FUNCTION_BLOCK FB_Syntax_ExhaustiveArraysAndFBInit
VAR
    // --- 1. Basic & Multi-dimensional Arrays ---
    arr1DPrimitives      : ARRAY[1..5] OF INT := [10, 20, 30, 40, 50];
    arr1DMultilineMatrix : ARRAY[1..12] OF INT := [
        1, 2, 3, 4,
        5, 6, 7, 8,
        9, 10, 11, 12
    ];
    arr2DMatrix : ARRAY[1..3, 1..4] OF INT;
    arr3DCube   : ARRAY[0..1, 0..1, 0..1] OF BOOL;
    arr4DHyper  : ARRAY[1..2, 1..2, 1..2, 1..2] OF BYTE;

    // --- 2. Negative, Zero-based, and Subrange Bounds ---
    arrNegativeBounds : ARRAY[-5..5] OF INT     := [-5, -4, -3, -2, -1, 0, 1, 2, 3, 4, 5];
    arrOffsetBounds   : ARRAY[100..105] OF DINT := [1000, 1001, 1002, 1003, 1004, 1005];

    // --- 3. Repetition / Initialization Factors ---
    arrRepeatZeros  : ARRAY[1..100] OF INT      := [100(0)];
    arrRepeatMixed  : ARRAY[1..10] OF INT       := [5(15), 3(25), 2(0)];
    arrRepeatString : ARRAY[1..4] OF STRING(30) := [2('READY'), 2('ERROR')];

    // --- 4. Arrays of STRUCT / UDT ---
    arrStructSingleLine     : ARRAY[1..4] OF ST_Syntax_Mini := [
        (nId := 1, bActive := TRUE, sName := 'Stage-Inlet'),
        (nId := 2, bActive := TRUE, sName := 'Stage-Reaction'),
        (nId := 3, bActive := TRUE, sName := 'Stage-Separation'),
        (nId := 4, bActive := TRUE, sName := 'Stage-Outlet')
    ];
    arrStructExpanded       : ARRAY[1..2] OF ST_Syntax_Mini := [
        (
            nId     := 101,
            bActive := TRUE,
            sName   := 'NodeA'
        ),
        (
            nId     := 102,
            bActive := FALSE,
            sName   := 'NodeB'
        )
    ];

    // --- 5. Arrays of Function Blocks with FB_init Parameters ---
    arrFbInitSingleLine : ARRAY[1..2] OF FB_Syntax_FBInitMethods[(nInitialId := 1, sInitialName := 'MotorA'), (nInitialId := 2, sInitialName := 'MotorB')];
    arrFbInitMultiline  : ARRAY[1..2] OF FB_Syntax_FBInitMethods[(nInitialId := 10, sInitialName := 'Sensor_Primary'), (nInitialId := 20, sInitialName := 'Sensor_Secondary')];

    // --- 6. Arrays of POINTER TO and INTERFACE ---
    arrPointers       : ARRAY[1..4] OF POINTER TO DINT;
    arrStructPointers : ARRAY[1..4] OF POINTER TO ST_Syntax_Mini;
    arrInterfaces     : ARRAY[1..4] OF I_Syntax_BaseDevice;

    // --- 7. Matrix with Row Comments ---
    arrMatrixCommented      : ARRAY[1..9] OF INT := [
        10, 5, 0, // Row 1
        5, 10, 5, // Row 2
        0, 5, 10  // Row 3
    ];

    // --- 8. Working variables ---
    nLoopIdx   : INT;
    nMatrixSum : DINT := 0;
END_VAR

// Matrix calculations
nMatrixSum   := 0;

FOR nLoopIdx := 1 TO 3 DO
    nMatrixSum := nMatrixSum + arr2DMatrix[nLoopIdx, 1];
END_FOR

// Array assignments and access
arr1DPrimitives[1]             := arr1DPrimitives[2] + arr1DPrimitives[3];
arr3DCube[0, 1, 0]             := NOT arr3DCube[1, 0, 1];
arrStructSingleLine[1].bActive := TRUE;
arrStructExpanded[1].nId       := 105;

// Interface check
IF arrInterfaces[1] <> 0 THEN
    arrInterfaces[1].M_Start(bForce := TRUE);
END_IF

END_FUNCTION_BLOCK

(* stored: Version 1.1.0.1, ProductVersion 3.1.4024.16
   POU FB_Syntax_ExhaustiveArraysAndFBInit: Id {a5d8924b-3c1e-450f-923f-e89c6239bc71}, SpecialFunc None *)
